// TIA Portal V21 export
ORGANIZATION_BLOCK "Main"   // OB1, LAD, ProgramCycle
TITLE = "Main Program Sweep (Cycle)"
{ S7_Optimized_Access := 'TRUE' }
// stored: SetENOAutomatically false
   VAR_INPUT
      Initial_Call : Bool;   // Initial call of this OB
      Remanence : Bool;   // =True, if remanent data are available
   END_VAR
BEGIN

REGION Network 1
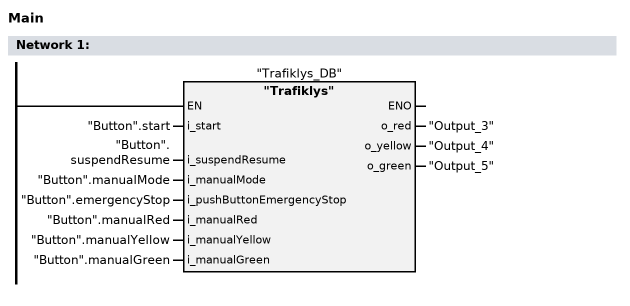
   RUNG wire#powerrail
      "Trafiklys_DB"(i_start := "Button".start, i_suspendResume := "Button".suspendResume, i_manualMode := "Button".manualMode, i_pushButtonEmergencyStop := "Button".emergencyStop, i_manualRed := "Button".manualRed, i_manualYellow := "Button".manualYellow, i_manualGreen := "Button".manualGreen, o_red => "Output_3", o_yellow => "Output_4", o_green => "Output_5")
   END_RUNG
   // the same network as SCL:
   "Trafiklys_DB"(i_start := "Button".start,   // "Trafiklys"
                  i_suspendResume := "Button".suspendResume,
                  i_manualMode := "Button".manualMode,
                  i_pushButtonEmergencyStop := "Button".emergencyStop,
                  i_manualRed := "Button".manualRed,
                  i_manualYellow := "Button".manualYellow,
                  i_manualGreen := "Button".manualGreen,
                  o_red => "Output_3",
                  o_yellow => "Output_4",
                  o_green => "Output_5");
END_REGION

REGION Network 3 (SCL)
   "Button".start := "Input_0";
   "Button".suspendResume := "Input_1";
   "Button".manualMode := "Input_2";
   "Button".emergencyStop := "Input_3";
   "Button".manualRed := "Input_4";
   "Button".manualYellow := "Input_5";
   "Button".manualGreen := "Input_6";
END_REGION
END_ORGANIZATION_BLOCK
